FUNCTION F_ConvertZisterne_mA2Perc : INT
VAR_INPUT
	i_Value			:	INT;
END_VAR
VAR_OUTPUT
END_VAR
VAR
	i_finalValue	:	INT;
	r_converted		:	REAL;
END_VAR

r_converted := (INT_TO_REAL(i_Value) / 200);

i_finalValue := REAL_TO_INT(r_converted * 100);

IF i_finalValue > 100 THEN
	i_finalValue := 100;
END_IF

F_ConvertZisterne_mA2Perc := i_finalValue;

END_FUNCTION

(* stored: Version 1.1.0.1, ProductVersion 3.1.4024.4
   POU F_ConvertZisterne_mA2Perc: Id {b0156247-7874-4cd0-86e5-a8806e84d105}, SpecialFunc None *)
